// TIA Portal V18 export
TYPE "HMI_Axis"
   STRUCT
      INPUT : Struct
         Axis_ID : Int := 1;   // 伺服ID
         Speed : Int;   // 伺服速度
         SimplyTrigger : Bool;   // 直接启动
         ListTrigger : Bool;   // 位置列表启动
         ListPosID : Int;   // 位置列表位置ID
         SimplyPos : Real;   // 直接启动位置
         Enable : Bool;   // 使能
         "Jog+" : Bool;
         "Jog-" : Bool;
         Homing : Bool;   // 回零
         Stop : Bool;   // 暂停
      END_STRUCT;
      OUTPUT : Struct
         Ready : Bool;   // 准备OK显示
         Alarm : Bool;   // 报警显示
         Warming : Bool;   // 警告显示
         RunEnd : Bool;   // 运行结束显示
         Interference : Bool;   // 干涉条件显示
         "Reference Point" : Bool;   // 参考点存在显示
         CurrentPosition : Real;   // 当前位置显示
         CurrentSpeed : Real;   // 当前速度显示
         TargetPosition : Real;   // 目标位置
         Enable : Bool;   // 使能显示
         MAX_Axis : Int := 1;
      END_STRUCT;
   END_STRUCT;
END_TYPE
